DATA_BLOCK "ifbHMISelectBLK_DB"
{ S7_Optimized_Access := 'TRUE' }
VERSION : 0.1
NON_RETAIN
"ifbHMISelectBLK"

BEGIN

END_DATA_BLOCK

